FUNCTION_BLOCK E_MERGE_3 (* Composite Function Block Type *)
  (* Standard: 61499-2 *)
  (* Version 0.0, 2018-11-02, 4DIAC-IDE, 4DIAC-Consortium *)
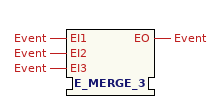
  EVENT_INPUT
    EI1;
    EI2;
    EI3;
  END_EVENT
  EVENT_OUTPUT
    EO;
  END_EVENT
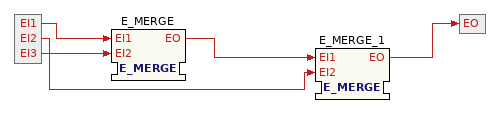
  FBS
    E_MERGE : E_MERGE;
    E_MERGE_1 : E_MERGE;
  END_FBS
  EVENT_CONNECTIONS
    EI1 TO E_MERGE.EI1;
    EI2 TO E_MERGE.EI2;
    E_MERGE.EO TO E_MERGE_1.EI1;
    EI3 TO E_MERGE_1.EI2;
    E_MERGE_1.EO TO EO;
  END_CONNECTIONS
END_FUNCTION_BLOCK
